{attribute 'qualified_only'}
{attribute 'strict'}
TYPE EFeedbackMsgSJH108 :
(
	StateMsg := 1,
	StatusMsg := 2,
	IsAliveMsg := 3,
	AlarmMsg := 10,
	AirValveIsOpenMsg,
	StaticEliminationInterruptMsg,
	RefreshingMsg
);
END_TYPE

(* stored: Version 1.1.0.1, ProductVersion 3.1.4024.12
   DUT EFeedbackMsgSJH108: Id {9d7b7e6d-7ed0-4634-8980-1321c8b96b88} *)
